// TwinCAT 3 PLC project Test
// ProgramVersion: 3.1.4026.16
// libraries:
//   Tc2_Standard, * (Beckhoff Automation GmbH)
//   Tc2_System, * (Beckhoff Automation GmbH)
//   StageCore, * (_)
//   StageUtils, * (_)
// project tree:
//   Broadcast Test/ TestCall.TcPOU, Test_Broadcast_FillAndCoalesce.TcPOU, Test_Broadcast_FillAndMove.TcPOU
//   EC Tests/ Test_Ec_CompCast.TcPOU, Test_Ec_FillAndMove.TcPOU, Test_Ec_FillAndCoalesce.TcPOU (not stored)
//   / MAIN.TcPOU, PlcTask.TcTTO
//   Strings/ Test_Strings_WildcardCmp.TcPOU
// (motion and I/O tree: see PLC project stageutils)
// real-time tasks:
//   TASK Example: cycle T#10ms, priority 20, ADS port 350
//   TASK Test: cycle T#10ms, priority 21, ADS port 351
//   TASK VISU_TASK: cycle T#200000us, priority 30, ADS port 352

CONFIGURATION Test
    RESOURCE PLC ON TwinCAT3
        TASK PlcTask(INTERVAL := T#10ms, PRIORITY := 21);
        PROGRAM MAIN WITH PlcTask : MAIN;
    END_RESOURCE
END_CONFIGURATION

// ---- MAIN.TcPOU
PROGRAM MAIN
VAR
	//ec_test_01				: Test_Ec_FillAndMove;
	//ec_test_02				: Test_Ec_FillAndCoalesce;
	//ec_test_03				: Test_Ec_CompCast;
	
	broadcast_test_01		: Test_Broadcast_FillAndMove;
	broadcast_test_02		: Test_Broadcast_FillAndCoalesce;
	
	strings_test_01			: Test_Strings_WildcardCmp;

	debugInfo				: StageCore.DebugInfo;
	
END_VAR

Runtime();

END_PROGRAM

// ---- Broadcast Test/Test_Broadcast_FillAndMove.TcPOU
// ASSUME Param.COMP_CAP = 20
// Fills _Ec.comp table with first batch of signals
// Then fills _Ec.comp table with second batch of signals.
// Entity 1 components need to be moved to the end, _Ec.iFirst is now Entity 2.
// Entity 2 components expand towards the position 1.
// Entity 3 components need to be moved to the end.
// At the end the entity range should be number of compoennets plus header.
FUNCTION_BLOCK Test_Broadcast_FillAndMove IMPLEMENTS I_Execute
VAR_INPUT
	bTest		: BOOL;
END_VAR
VAR_OUTPUT
(*
	Resulting _Ec.comp table:
	1. EMPTY
	2. Signal[2] - Header
	3. batch02[2, 2]
	4. batch02[2, 1]
	5. batch01[2, 1]
	6. batch01[2, 2]
	7. EMPTY
	8. EMPTY
	9. EMPTY
	10. Signal[1] - Header
	11. batch01[1, 1]
	12. batch01[1, 2]
	13. batch02[1, 1]
	14. batch02[1, 2]
	15. Signal[3] - Header
	16. batch01[3, 1]
	17. batch01[3, 2]
	18. batch02[3, 1]
	19. batch02[3, 2]
	20. EMPTY
*)
END_VAR
VAR
	exe					: Execute(THIS^);	
	call				: TestCall;

	signal				: ARRAY[1..3] OF Signal; // 3 headers
	
	batch01				: ARRAY[1..3, 1..2] OF Receiver(call); // 6 entries
	batch02				: ARRAY[1..3, 1..2] OF Receiver(call);	// another 6 entries
	
	i, j				: UDINT;
END_VAR

METHOD Execute
IF bTest THEN
	FOR i := 1 TO 3 DO
		FOR j := 1 TO 2 DO
			signal[i].Pair(batch01[i, j]);
		END_FOR
	END_FOR

	FOR i := 1 TO 3 DO
		FOR j := 1 TO 2 DO
			signal[i].Pair(batch02[i, j]);
		END_FOR
	END_FOR

	bTest := FALSE;
END_IF
END_METHOD

END_FUNCTION_BLOCK

// ---- Broadcast Test/TestCall.TcPOU
FUNCTION_BLOCK TestCall IMPLEMENTS I_Callable
VAR_INPUT
END_VAR
VAR_OUTPUT
END_VAR
VAR
	nUdint		: UDINT;
END_VAR

METHOD Call
VAR_INPUT
	iArg	: Core.I_Arg;
END_VAR
nUdint := nUdint + 1;
END_METHOD

END_FUNCTION_BLOCK

// ---- Broadcast Test/Test_Broadcast_FillAndCoalesce.TcPOU
// ASSUME Param.COMP_CAP = 20
// Fills _Ec.comp table with first batch of signals
// Then fills _Ec.comp table with second batch of signals.
// Entity 1 components need to be moved to the end, _Ec.iFirst is now Entity 2.
// Entity 2 components expand towards the position 1.
// Entity 3 components need to be moved to the end.

// Fill _Ec.comp with 3rd batch of signals forcing table to coalesce

// At the end the entity range should be number of compoennets plus header.
FUNCTION_BLOCK Test_Broadcast_FillAndCoalesce IMPLEMENTS I_Execute
VAR_INPUT
	bTest		: BOOL;
END_VAR
VAR_OUTPUT
(*
	Resulting _Ec.comp table:
	1. Signal[1] - Header
	2. batch01[1, 1]
	3. batch01[1, 2]
	4. batch02[1, 1]
	5. batch02[1, 2]
	6. Signal[2] - Header
	7. batch02[2, 2]
	8. batch02[2, 1]
	9. batch01[2, 1]
	10. batch01[2, 2]
	11. Signal[3] - Header
	12. batch01[3, 1]
	13. batch02[3, 2]
	14. batch02[3, 1]
	15. batch01[3, 2]
	16. CoalSignal - Header
	17. coalBatch[1]
	18. coalBatch[2]
	19. coalBatch[3]
	20. EMPTY
*)
END_VAR
VAR
	exe					: Execute(THIS^);	
	call				: TestCall;

	signal				: ARRAY[1..3] OF Signal; // 3 headers
	dfgSignal			: Signal;
	
	batch01				: ARRAY[1..3, 1..2] OF Receiver(call); // 6 entries
	batch02				: ARRAY[1..3, 1..2] OF Receiver(call);	// another 6 entries
	dfgBatch			: ARRAY[1..4] OF Receiver(call);
	
	i, j				: UDINT;
END_VAR

METHOD Execute
VAR_INPUT
	nPhase: INT := 0;
END_VAR
IF bTest THEN
	FOR i := 1 TO 3 DO
		FOR j := 1 TO 2 DO
			signal[i].Pair(batch01[i, j]);
		END_FOR
	END_FOR

	FOR i := 1 TO 3 DO
		FOR j := 1 TO 2 DO
			signal[i].Pair(batch02[i, j]);
		END_FOR
	END_FOR
	
	FOR i := 1 TO 4 DO
		dfgSignal.Pair(dfgBatch[i]);
	END_FOR

	bTest := FALSE;
END_IF
END_METHOD

END_FUNCTION_BLOCK

// ---- Strings/Test_Strings_WildcardCmp.TcPOU
FUNCTION_BLOCK Test_Strings_WildcardCmp IMPLEMENTS I_Execute
VAR_INPUT
	bTest			: BOOL;
END_VAR
VAR_OUTPUT
	nMatchResult	: USINT;
END_VAR
VAR
	exe				: Execute(THIS^);
	sAddress		: Str := 'abc.def.ghi.jkl';
	sPattern		: ARRAY[1..10] OF Str := ['abc.def.ghi.jkl', 'abc.*', '*.ghi.*', '*.ghi', '*.jkl.*', 'abc.*.*.jkl', 'abc.*.*.*', 'abc.def.xyz.jkl', 'abc.def', '*'];
	nResult			: ARRAY[1..10] OF Result;
	nExpected		: ARRAY[1..10] OF Result := [Ok, Ok, Ok, None, Ok, Ok, Ok, None, None, Ok];
	i				: USINT;
END_VAR

METHOD Execute
IF bTest THEN
	FOR i := 1 TO 10 DO
		nResult[i] := MatchTagPathPattern(sAddress, sPattern[i]);
		IF nResult[i] = nExpected[i] THEN
			nMatchResult := nMatchResult + 1;
		END_IF
	END_FOR	

	bTest := FALSE;
END_IF
END_METHOD

END_FUNCTION_BLOCK

// ---- EC Tests/Test_Ec_CompCast.TcPOU
// ASSUME Param.COMP_CAP = 20
// Fills _Ec.comp table with first batch of signals
// Then fills _Ec.comp table with second batch of signals.
// Entity 1 components need to be moved to the end, _Ec.iFirst is now Entity 2.
// Entity 2 components expand towards the position 1.
// Entity 3 components need to be moved to the end.

// Fill _Ec.comp with 3rd batch of signals forcing table to coalesce

// At the end the entity range should be number of compoennets plus header.
FUNCTION_BLOCK Test_Ec_CompCast IMPLEMENTS I_Execute
VAR_INPUT
	bTest				: BOOL;
END_VAR
VAR_OUTPUT
	iTag				: I_Tag;
	iSignal				: I_Signal;
	iState				: I_State;
END_VAR
VAR
	exe					: Execute(THIS^);	
	
	tag					: Tag('Casting test');	
	iComp				: I_Component := tag;
	
	
	i, j				: UDINT;
END_VAR

METHOD Execute
IF bTest THEN
	Core.CompAsITag(iComp, iDest => iTag);
	Core.CompAsIState(iComp, iDest => iState);
	Core.CompAsISignal(iComp, iDest => iSignal);

	bTest := FALSE;
END_IF
END_METHOD

END_FUNCTION_BLOCK

// ---- EC Tests/Test_Ec_FillAndMove.TcPOU
// ASSUME Param.COMP_CAP = 20
// Fills _Ec.comp table with first batch of signals
// Then fills _Ec.comp table with second batch of signals.
// Entity 1 components need to be moved to the end, _Ec.iFirst is now Entity 2.
// Entity 2 components expand towards the position 1.
// Entity 3 components need to be moved to the end.
// At the end the entity range should be number of compoennets plus header.
FUNCTION_BLOCK Test_Ec_FillAndMove IMPLEMENTS I_Execute
VAR_INPUT
	bTest		: BOOL;
END_VAR
VAR_OUTPUT
(*
	Resulting _Ec.comp table:
	1. EMPTY
	2. Entity[2] - Header
	3. batch02[2, 2]
	4. batch02[2, 1]
	5. batch01[2, 1]
	6. batch01[2, 2]
	7. EMPTY
	8. EMPTY
	9. EMPTY
	10. Entity[1] - Header
	11. batch01[1, 1]
	12. batch01[1, 2]
	13. batch02[1, 1]
	14. batch02[1, 2]
	15. Entity[3] - Header
	16. batch01[3, 1]
	17. batch01[3, 2]
	18. batch02[3, 1]
	19. batch02[3, 2]
	20. EMPTY
*)
END_VAR
VAR
	exe					: Execute(THIS^);	

	entity				: ARRAY[1..3] OF Entity; // 3 headers
	
	batch01				: ARRAY[1..3, 1..2] OF Signal; // 6 entries
	batch02				: ARRAY[1..3, 1..2] OF Signal;	// another 6 entries
	
	i, j				: UDINT;
END_VAR

METHOD Execute
IF bTest THEN
	FOR i := 1 TO 3 DO
		FOR j := 1 TO 2 DO
			RegComp(batch01[i, j], entity[i]);
		END_FOR
	END_FOR

	FOR i := 1 TO 3 DO
		FOR j := 1 TO 2 DO
			RegComp(batch02[i, j], entity[i]);
		END_FOR
	END_FOR

	bTest := FALSE;
END_IF
END_METHOD

END_FUNCTION_BLOCK
